FUNCTION_BLOCK PUBLIC FacadePrinterNormal
VAR_INPUT
END_VAR
VAR_OUTPUT
END_VAR
VAR
	printer :  Printer;
END_VAR

METHOD FB_init : BOOL
VAR_INPUT
	bInitRetains : BOOL; // if TRUE, the retain variables are initialized (warm start / cold start)
	bInCopyCode : BOOL;  // if TRUE, the instance afterwards gets moved into the copy code (online change)
	text : STRING;
	color : BOOL;
	sheet : STRING;
	documentType : STRING;
	
END_VAR

printer.setColor(color);
printer.setSheet(sheet);
printer.setdocumentType(documentType);
printer.setText(text);
END_METHOD

METHOD print
printer.printDocument();
END_METHOD

END_FUNCTION_BLOCK

(* stored: Version 1.1.0.1, ProductVersion 3.1.4024.12
   POU FacadePrinterNormal: Id {52c24485-e01b-4331-8859-a3576c7ec019}, SpecialFunc None
   Method FB_init: Id {7b799386-3fd5-476f-b8cb-3301efd26b63}
   Method print: Id {35024de5-e274-42d1-962d-b021b9a478b5} *)
